{attribute 'enable_dynamic_creation'}
FUNCTION_BLOCK CMD_RemoteMode IMPLEMENTS I_Command
VAR_INPUT
END_VAR
VAR_OUTPUT
END_VAR
VAR
	Comms : I_CommsTransmitter;
	Status : (IDLE, EXECUTE, SENDING, SENT, COMPLETE, TIMED_OUT);
	WatchDog : WatchDog; 
END_VAR
VAR CONSTANT
	CMD : STRING := 'SYSTem:REMote$R$N';
	TIME_OUT : TIME := T#2S;	
END_VAR

CASE Status OF
	
	EXECUTE: 
		WatchDog.Enable(TIME_OUT);
		Status := SENDING;
		
	SENDING:
		IF Comms.isBusy THEN
			RETURN;
		ELSE
			Comms.Send(CMD);
			Status := SENT;
		END_IF
		
	SENT:
		IF Comms.isBusy THEN
			RETURN;
		ELSE
			WatchDog.Disable();
			Status := COMPLETE;
		END_IF

	IDLE: //
	COMPLETE://
	TIMED_OUT: //
	
END_CASE

IF WatchDog.isTriggered THEN
	WatchDog.Disable();
	Status := TIMED_OUT;
END_IF

METHOD Destroy
VAR_INPUT
END_VAR
VAR
	selfPointer: POINTER TO CMD_RemoteMode;
END_VAR
selfPointer := ADR(THIS^);
__DELETE(selfPointer);
END_METHOD

METHOD PUBLIC Execute : BOOL
VAR_INPUT
END_VAR
IF NOT isBusy THEN
	Status := EXECUTE;
	Execute := TRUE;
END_IF

THIS^();
END_METHOD

METHOD FB_init : BOOL
VAR_INPUT
	bInitRetains : BOOL; // if TRUE, the retain variables are initialized (warm start / cold start)
	bInCopyCode : BOOL;  // if TRUE, the instance afterwards gets moved into the copy code (online change)
	Comms : I_CommsTransmitter;
END_VAR
THIS^.Comms := Comms;
END_METHOD

PROPERTY PUBLIC hasTimedOut : BOOL
GET
hasTimedOut := (Status = TIMED_OUT) ;
END_GET
END_PROPERTY

PROPERTY PUBLIC isBusy : BOOL
GET
isBusy := not (Status = IDLE or Status = COMPLETE or Status = TIMED_OUT);
END_GET
END_PROPERTY

PROPERTY isComplete : BOOL
GET
isComplete := (Status = COMPLETE or Status = TIMED_OUT) ;
END_GET
END_PROPERTY

END_FUNCTION_BLOCK

(* stored: Version 1.1.0.1, ProductVersion 3.1.4024.9
   POU CMD_RemoteMode: Id {693695f4-74f5-4119-90c6-9c642ed01ec9}, SpecialFunc None
   Method Destroy: Id {fc2d226b-dfbd-4242-8aac-4ae4555b8d82}
   Method Execute: Id {b0b43112-947c-4a55-812d-aad2066cf74a}
   Method FB_init: Id {01320c37-2820-4e5b-97d0-f91acb46a19b}
   Property hasTimedOut: Id {857ca9e9-914b-44ab-936f-e6f28df148fc}
   Get Get: Id {0b98c16a-774e-4308-882b-fe0b1847e759}
   Property isBusy: Id {2cc21b9e-e7d3-4dc1-8322-c3834ceb937b}
   Get Get: Id {06554164-0ad3-4d3b-9d20-0af5f609e2dc}
   Property isComplete: Id {40efd645-d133-4c4e-a968-d2d464fb9529}
   Get Get: Id {9a045034-bdc0-4549-8599-b5a3cde73040} *)
